//执行完一次iFileState循环后，控制器UsrData文件夹内有test2.txt文件，需要删除之后才能再次循环，否则重命名时因文件名已存在会报错	  
IF restart THEN
   DelFileName :='/usr/src/CODESYSControl/UsrData/test2.txt';
   xFileDelete:=TRUE;
   TON_2(IN:= xFileDelete, PT:= T#100MS, Q=> , ET=> );  //删除文件延时判断
      IF TON_2.Q THEN
		  IF FileDeleteErrorID = 0 THEN 
             xFileDelete :=FALSE;
             TON_2(IN:= xFileDelete, PT:= T#10MS, Q=> , ET=> );  //复位定时器
			 restart:=FALSE;
			 iFileState:=1;
			ELSE  xFileDelete:=FALSE;
                  iFileState:=10;
				  RETURN; 
		  END_IF  
	  END_IF 
END_IF         
END_CASE

ACTION ACT_SysFileRead:
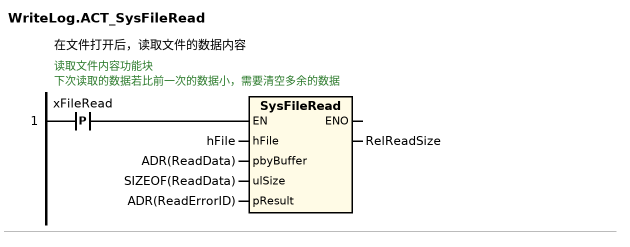
// NETWORK 1: 在文件打开后，读取文件的数据内容
// 读取文件内容功能块
// 下次读取的数据若比前一次的数据小，需要清空多余的数据
_rt1(CLK := xFileRead);
IF _rt1.Q THEN
    RelReadSize := SysFileRead(hFile := hFile, pbyBuffer := ADR(ReadData), ulSize := SIZEOF(ReadData), pResult := ADR(ReadErrorID));
END_IF
END_ACTION

ACTION ACT_SysFileDelete:
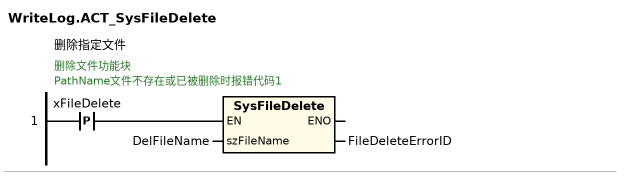
// NETWORK 1: 删除指定文件
// 删除文件功能块
// PathName文件不存在或已被删除时报错代码1
_rt2(CLK := xFileDelete);
IF _rt2.Q THEN FileDeleteErrorID := SysFileDelete(szFileName := DelFileName); END_IF
END_ACTION

ACTION ACT_SysFileClose:
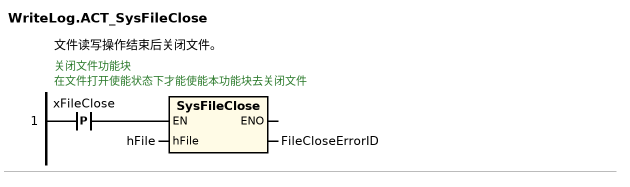
// NETWORK 1: 文件读写操作结束后关闭文件。
// 关闭文件功能块
// 在文件打开使能状态下才能使能本功能块去关闭文件
_rt3(CLK := xFileClose);
IF _rt3.Q THEN FileCloseErrorID := SysFileClose(hFile := hFile); END_IF
END_ACTION

ACTION ACT_SysFileRename:
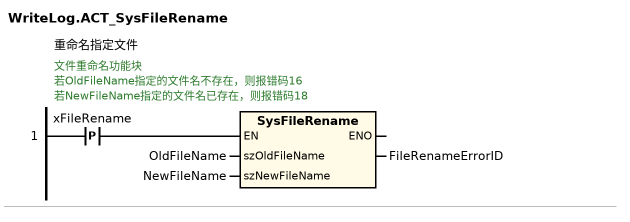
// NETWORK 1: 重命名指定文件
// 文件重命名功能块
// 若OldFileName指定的文件名不存在，则报错码16
// 若NewFileName指定的文件名已存在，则报错码18
_rt4(CLK := xFileRename);
IF _rt4.Q THEN
    FileRenameErrorID := SysFileRename(szOldFileName := OldFileName, szNewFileName := NewFileName);
END_IF
END_ACTION

ACTION ACT_SysFileGetPos:
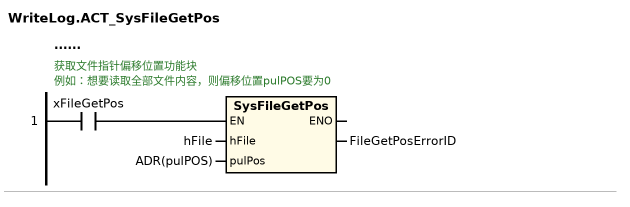
// NETWORK 1: ......
// 获取文件指针偏移位置功能块
// 例如：想要读取全部文件内容，则偏移位置pulPOS要为0
IF xFileGetPos THEN FileGetPosErrorID := SysFileGetPos(hFile := hFile, pulPos := ADR(pulPOS)); END_IF
END_ACTION

ACTION ACT_SysFileCopy:
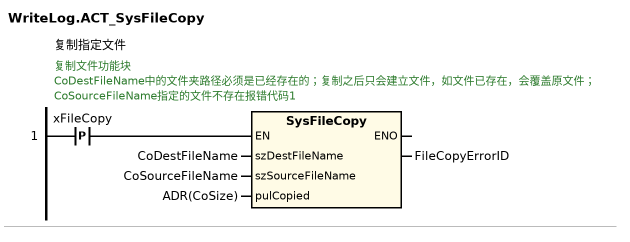
// NETWORK 1: 复制指定文件
// 复制文件功能块
// CoDestFileName中的文件夹路径必须是已经存在的；复制之后只会建立文件，如文件已存在，会覆盖原文件；
// CoSourceFileName指定的文件不存在报错代码1
_rt5(CLK := xFileCopy);
IF _rt5.Q THEN
    FileCopyErrorID := SysFileCopy(szDestFileName := CoDestFileName, szSourceFileName := CoSourceFileName, pulCopied := ADR(CoSize));
END_IF
END_ACTION

ACTION ACT_SysFileSetPos:
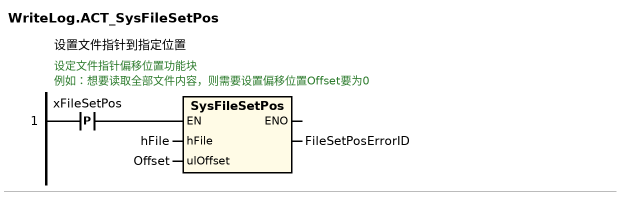
// NETWORK 1: 设置文件指针到指定位置
// 设定文件指针偏移位置功能块
// 例如：想要读取全部文件内容，则需要设置偏移位置Offset要为0
_rt6(CLK := xFileSetPos);
IF _rt6.Q THEN FileSetPosErrorID := SysFileSetPos(hFile := hFile, ulOffset := Offset); END_IF
END_ACTION

ACTION ACT_SysFileEOF:
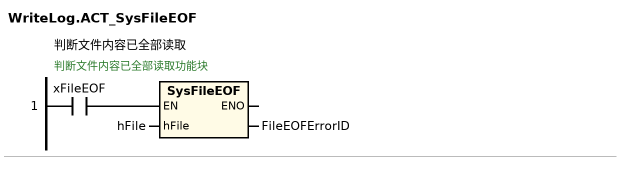
// NETWORK 1: 判断文件内容已全部读取
// 判断文件内容已全部读取功能块
IF xFileEOF THEN FileEOFErrorID := SysFileEOF(hFile := hFile); END_IF
END_ACTION

ACTION ACT_SysFileWrite:
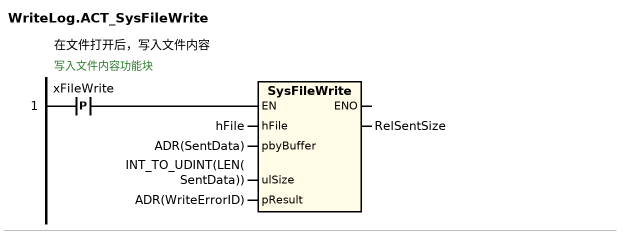
// NETWORK 1: 在文件打开后，写入文件内容
// 写入文件内容功能块
_rt7(CLK := xFileWrite);
IF _rt7.Q THEN
    RelSentSize := SysFileWrite(hFile := hFile, pbyBuffer := ADR(SentData), ulSize := INT_TO_UDINT(LEN(SentData)), pResult := ADR(WriteErrorID));
END_IF
END_ACTION

ACTION ACT_SysFileOpen:
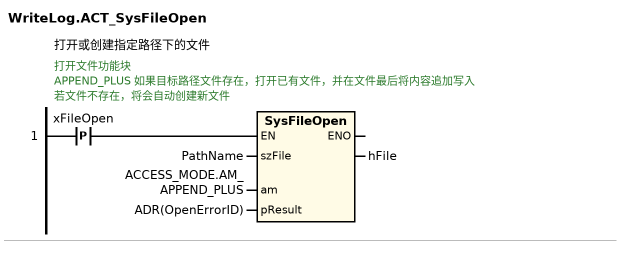
// NETWORK 1: 打开或创建指定路径下的文件
// 打开文件功能块
// APPEND_PLUS 如果目标路径文件存在，打开已有文件，并在文件最后将内容追加写入
//             若文件不存在，将会自动创建新文件
_rt8(CLK := xFileOpen);
IF _rt8.Q THEN
    hFile := SysFileOpen(szFile := PathName, am := ACCESS_MODE.AM_APPEND_PLUS, pResult := ADR(OpenErrorID));
END_IF
END_ACTION

END_PROGRAM

// Device/Application/BasicFBs/MeanValue
FUNCTION_BLOCK MeanValue
VAR_EXTERNAL

END_VAR

VAR_INPUT
	Input:UINT;
	PAR_Lenght:UINT;
	Reset:BOOL;
END_VAR
VAR_OUTPUT
	Output:UINT;
END_VAR
VAR
	Ka_Count:UINT:=1;
	Ka:UINT:=1;
	Ka_prev:UINT;
END_VAR

(*======================== READ_ME ==============================*)
(*功能块：“平均值滤波”                                         *)
(*=========================== END ===============================*)
	Ka:=UDINT_TO_UINT((UINT_TO_UDINT(Ka)*UINT_TO_UDINT(Ka_Count-1)+UINT_TO_UDINT(Input))/UINT_TO_UDINT(Ka_Count));
	Ka_Count:=Ka_count+1;
	IF(Reset OR Ka_count=PAR_Lenght+1) THEN
		Output:=Ka;
		Ka_Count:=1;
		Ka:=1;
	END_IF;

END_FUNCTION_BLOCK

// Device/Application/BasicFBs/Cut
FUNCTION_BLOCK Cut     (*把输入值进行预处理，调整斜率，消除两端的非线性影响*)
VAR_INPUT
	Input:UINT;
	PAR_InputlLowLimit:UINT;               (*此值的取值范围为0-255，一般在0—50之间*)
	PAR_InputHighLimit:UINT;               (*此值的取值范围为0-255，一般在200-255之间*)
END_VAR
VAR_OUTPUT
	Output:UINT;
	LowLimit:BOOL;
	HighLimit:BOOL;
END_VAR
VAR
END_VAR

(*功能描述：
把输入值进行预处理，调整斜率，消除两端非线性影响。
输入参数：
（1）Input，UINT型，要处理的信号。
（2）PAR_InputILowLimit，UINT型，用来控制输出的下限。当Input<=256*PAR_InputILowLimit时输出为0。
（3）PAR_InputHighLimit，UINT型，用来控制输出的上限。当Input>=256*PAR_InputHighLimit时输出就为256*PAR_InputHighLimit。
输出参数：
（1）Output，UINT型，处理完的信号。
（2）LowLimit，BOOL型，Input<=256*PAR_InputILowLimit时LowLimit为TRUE。
（3）HighLimit，BOOL型，Input>=256*PAR_InputHighLimit时HighLimit为TRUE。
*)

	LowLimit:=0;
	HighLimit:=0;
	PAR_InputlLowLimit:=PAR_InputlLowLimit*256;
	PAR_InputHighLimit:=PAR_InputHighLimit*256;
	IF(Input>=PAR_InputHighLimit) THEN
		Output:=0;
		HighLimit:=1;
	ELSIF(Input<=PAR_InputlLowLimit) THEN
		Output:=0;
		LowLimit:=1;
	ELSE
		Output:=DWORD_TO_UINT((Input-PAR_InputlLowLimit)*65536/(65536-PAR_InputlLowLimit-(65535-PAR_InputHighLimit)));
	END_IF

END_FUNCTION_BLOCK

// Device/Application/Motor
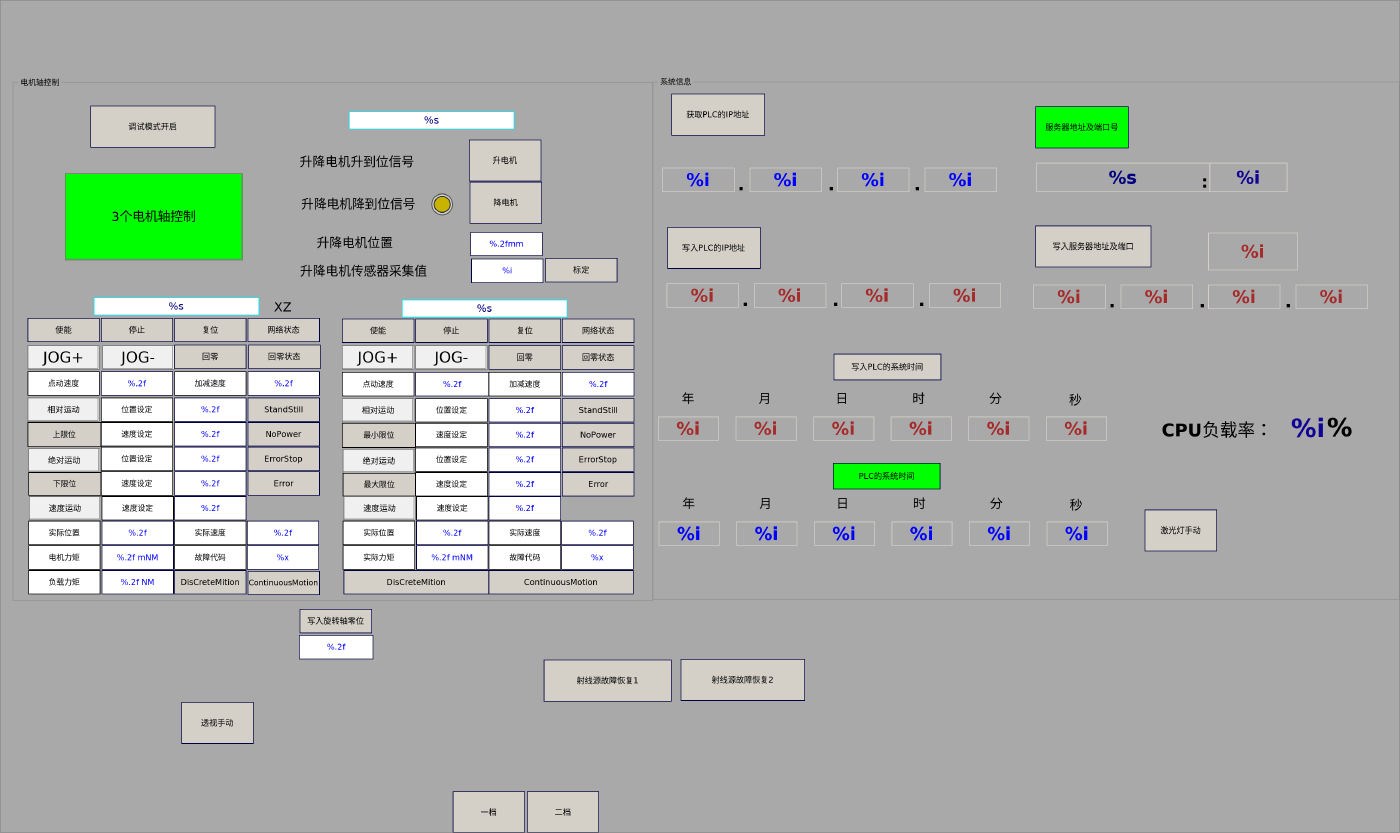
VISUALIZATION Motor  // 1985x1182
    Button (39,490 102x34), "JOG+", colour toggle: Axis_XZ.XZ_AxisCmd.bJogP
        tap Axis_XZ.XZ_AxisCmd.bJogP
    Rectangle (144,739 102x34), "%.2f", text variable: Axis_XZ.XZ_AxisState.rActPosition
    Button (145,490 102x34), "JOG-", colour toggle: Axis_XZ.XZ_AxisCmd.bJogN
        tap Axis_XZ.XZ_AxisCmd.bJogN
    RoundedRectangle (39,451 102x34), "使能", colour toggle: Axis_XZ.XZ_AxisState.bPowering
        toggle Axis_XZ.XZ_AxisCmd.bPower
    RoundedRectangle (351,451 102x34), "网络状态", colour toggle: Axis_XZ.XZ_AxisState.bNetState
    Button (40,636 102x34), "绝对运动", colour toggle: Axis_XZ.XZ_AxisCmd.bAbs
        tap Axis_XZ.XZ_AxisCmd.bAbs
    Rectangle (40,739 102x34), "实际位置"
    Rectangle (350,739 102x34), "%.2f", text variable: Axis_XZ.XZ_AxisState.rActVelocity
    Rectangle (247,739 102x34), "实际速度"
    RoundedRectangle (143,451 102x34), "停止", colour toggle: Axis_XZ.XZ_AxisState.bStopState
        tap Axis_XZ.XZ_AxisCmd.bStop
    RoundedRectangle (247,451 102x34), "复位", colour toggle: Axis_XZ.XZ_AxisCmd.bReset
        tap Axis_XZ.XZ_AxisCmd.bReset
    Rectangle (133,422 234x25), "%s", text variable: InitMotor.sNameXZ, text list: ''
    Rectangle (247,774 102x34), "故障代码"
    Rectangle (350,774 102x34), "%x", text variable: Axis_XZ.XZ_AxisState.ErrorID, colour toggle: (Axis_XZ.XZ_AxisState.ErrorID)<>0
    Rectangle (40,670 103x33), "下限位", colour toggle: Entity_IO.bRotateMotorMin
    Rectangle (39,599 104x35), "上限位", colour toggle: Entity_IO.bRotateMotorMax
    RoundedRectangle (247,489 102x34), "回零", colour toggle: Axis_XZ.XZ_AxisCmd.bHome
        tap Axis_XZ.XZ_AxisCmd.bHome
    Button (39,564 102x34), "相对运动", colour toggle: Axis_XZ.XZ_AxisCmd.bRel
        tap Axis_XZ.XZ_AxisCmd.bRel
    Rectangle (143,527 102x34), "%.2f", text variable: Axis_XZ.XZ_AxisCmd.AxisPara.rJogVelocity
        OnMouseClick: write Axis_XZ.XZ_AxisCmd.AxisPara.rJogVelocity via Default
    Rectangle (39,527 102x34), "点动速度"
    Rectangle (247,527 102x34), "加减速度"
    Rectangle (351,527 102x34), "%.2f", text variable: Axis_XZ.XZ_AxisCmd.AxisPara.rAccDec
        OnMouseClick: write Axis_XZ.XZ_AxisCmd.AxisPara.rAccDec via Default
    Rectangle (143,564 102x34), "位置设定"
    Rectangle (247,564 102x34), "%.2f", text variable: Axis_XZ.XZ_AxisCmd.AxisPara.rRelPosition
        OnMouseClick: write Axis_XZ.XZ_AxisCmd.AxisPara.rRelPosition via Default
    Rectangle (143,599 102x34), "速度设定"
    Rectangle (247,599 102x34), "%.2f", text variable: Axis_XZ.XZ_AxisCmd.AxisPara.rRelVelocity
        OnMouseClick: write Axis_XZ.XZ_AxisCmd.AxisPara.rRelVelocity via Default
    Rectangle (143,634 102x34), "位置设定"
    Rectangle (693,635 102x34), "%.2f", text variable: Axis_QJ.QJ_AxisCmd.AxisPara.rAbsPosition
        OnMouseClick: write Axis_QJ.QJ_AxisCmd.AxisPara.rAbsPosition via Default
    Rectangle (143,669 102x34), "速度设定"
    Rectangle (247,669 102x34), "%.2f", text variable: Axis_XZ.XZ_AxisCmd.AxisPara.rAbsVelocity
        OnMouseClick: write Axis_XZ.XZ_AxisCmd.AxisPara.rAbsVelocity via Default
    RoundedRectangle (351,564 102x34), "StandStill", colour toggle: Axis_XZ.XZ_AxisState.bStandStill
    RoundedRectangle (351,599 102x34), "NoPower", colour toggle: Axis_XZ.XZ_AxisState.bPowerOff
    RoundedRectangle (351,634 102x34), "ErrorStop", colour toggle: Axis_XZ.XZ_AxisState.bErrStop
    RoundedRectangle (351,669 102x34), "Error", colour toggle: Axis_XZ.XZ_AxisState.bAxisErr
    Rectangle (144,774 102x34), "%.2f mNM", text variable: Axis_XZ.XZ_AxisState.rActTorque
    Rectangle (40,774 102x34), "电机力矩"
    Rectangle (570,425 234x25), "%s", text variable: InitMotor.sNameQJ, text list: ''
    Button (485,490 102x34), "JOG+", colour toggle: Axis_QJ.QJ_AxisCmd.bJogP
        tap Axis_QJ.QJ_AxisCmd.bJogP
    Rectangle (590,739 102x34), "%.2f", text variable: Axis_QJ.QJ_AxisState.rActPosition
    Button (589,490 102x34), "JOG-", colour toggle: Axis_QJ.QJ_AxisCmd.bJogN
        tap Axis_QJ.QJ_AxisCmd.bJogN
    RoundedRectangle (485,452 102x34), "使能", colour toggle: Axis_QJ.QJ_AxisState.bPowering
        toggle Axis_QJ.QJ_AxisCmd.bPower
    RoundedRectangle (797,452 102x34), "网络状态", colour toggle: Axis_QJ.QJ_AxisState.bNetState
    Button (486,637 102x34), "绝对运动", colour toggle: Axis_QJ.QJ_AxisCmd.bAbs
        tap Axis_QJ.QJ_AxisCmd.bAbs
    Rectangle (486,739 102x34), "实际位置"
    Rectangle (796,739 102x34), "%.2f", text variable: Axis_QJ.QJ_AxisState.rActVelocity
    Rectangle (693,739 102x34), "实际速度"
    RoundedRectangle (589,452 102x34), "停止", colour toggle: Axis_QJ.QJ_AxisCmd.bStop
        tap Axis_QJ.QJ_AxisCmd.bStop
    RoundedRectangle (693,452 102x34), "复位", colour toggle: Axis_QJ.QJ_AxisCmd.bReset
        tap Axis_QJ.QJ_AxisCmd.bReset
    Rectangle (693,774 102x34), "故障代码"
    Rectangle (796,774 102x34), "%x", text variable: Axis_QJ.QJ_AxisState.ErrorID, colour toggle: (Axis_QJ.QJ_AxisState.ErrorID)<>0
    Rectangle (486,671 103x33), "最大限位", colour toggle: Entity_IO.bForeMotorMax
    Rectangle (485,600 104x35), "最小限位", colour toggle: Entity_IO.bForeMotorMin
    RoundedRectangle (693,490 102x34), "回零", colour toggle: Axis_QJ.QJ_AxisCmd.bHome
        tap Axis_QJ.QJ_AxisCmd.bHome
    Button (485,565 102x34), "相对运动", colour toggle: Axis_QJ.QJ_AxisCmd.bRel
        tap Axis_QJ.QJ_AxisCmd.bRel
    Rectangle (589,528 104x34), "%.2f", text variable: Axis_QJ.QJ_AxisCmd.AxisPara.rJogVelocity
        OnMouseClick: write Axis_QJ.QJ_AxisCmd.AxisPara.rJogVelocity via Default
    Rectangle (485,528 102x34), "点动速度"
    Rectangle (693,528 102x34), "加减速度"
    Rectangle (797,528 102x34), "%.2f", text variable: Axis_QJ.QJ_AxisCmd.AxisPara.rAccDec
        OnMouseClick: write Axis_QJ.QJ_AxisCmd.AxisPara.rAccDec via Default
    Rectangle (589,565 102x34), "位置设定"
    Rectangle (693,565 102x34), "%.2f", text variable: Axis_QJ.QJ_AxisCmd.AxisPara.rRelPosition
        OnMouseClick: write Axis_QJ.QJ_AxisCmd.AxisPara.rRelPosition via Default, min -1000, max 1000
    Rectangle (589,600 102x34), "速度设定"
    Rectangle (693,600 102x34), "%.2f", text variable: Axis_QJ.QJ_AxisCmd.AxisPara.rRelVelocity
        OnMouseClick: write Axis_QJ.QJ_AxisCmd.AxisPara.rRelVelocity via Default
    Rectangle (589,635 102x34), "位置设定"
    Rectangle (247,634 102x34), "%.2f", text variable: Axis_XZ.XZ_AxisCmd.AxisPara.rAbsPosition
        OnMouseClick: write Axis_XZ.XZ_AxisCmd.AxisPara.rAbsPosition via Default
    Rectangle (589,670 102x34), "速度设定"
    Rectangle (693,670 102x34), "%.2f", text variable: Axis_QJ.QJ_AxisCmd.AxisPara.rAbsVelocity
        OnMouseClick: write Axis_QJ.QJ_AxisCmd.AxisPara.rAbsVelocity via Default
    RoundedRectangle (797,565 102x34), "StandStill", colour toggle: Axis_QJ.QJ_AxisState.bStandStill
    RoundedRectangle (797,600 102x34), "NoPower", colour toggle: Axis_QJ.QJ_AxisState.bPowerOff
    RoundedRectangle (797,635 102x34), "ErrorStop", colour toggle: Axis_QJ.QJ_AxisState.bErrStop
    RoundedRectangle (797,670 102x34), "Error", colour toggle: Axis_QJ.QJ_AxisState.bAxisErr
    Rectangle (590,774 102x34), "%.2f mNM", text variable: Axis_QJ.QJ_AxisState.rActTorque
    Rectangle (486,774 102x34), "实际力矩"
    RoundedRectangle (487,809 206x34), "DisCreteMition", colour toggle: Axis_QJ.QJ_AxisState.bDisCreteMition
    RoundedRectangle (693,809 205x34), "ContinuousMotion", colour toggle: Axis_QJ.QJ_AxisState.bContinuousMotion
    RoundedRectangle (247,809 102x34), "DisCreteMition", colour toggle: Axis_XZ.XZ_AxisState.bDisCreteMition
    RoundedRectangle (351,810 102x34), "ContinuousMotion", colour toggle: Axis_XZ.XZ_AxisState.bContinuousMotion
    RoundedRectangle (128,150 177x59), "调试模式开启", colour toggle: WorkMode.bDebugMode
        toggle WorkMode.bDebugMode
    Rectangle (495,158 234x25), "%s", text variable: InitMotor.sNameSJ, text list: ''
    RoundedRectangle (665,198 102x59), "升电机", colour toggle: Entity_IO.bUpMotorPos
        tap Entity_IO.bUpMotorPos
    RoundedRectangle (666,258 102x59), "降电机", colour toggle: Entity_IO.bUpMotorNeg
        tap Entity_IO.bUpMotorNeg
    Label (410,212 192x36), "升降电机升到位信号"
    Label (412,272 192x36), "升降电机降到位信号"
    Lamp1 (608,272 38x36), variable: Entity_IO.bUpMotorMin, style: Lamp-Lamp1-Yellow
    Button (92,246 252x123), "3个电机轴控制"
        OnMouseClick:  Assign=Catalogue, Type=Assignment
    RoundedRectangle (773,366 102x34), "标定", colour toggle: Entity_IO.bCalibrate
        tap Entity_IO.bCalibrate
    Rectangle (667,329 102x34), "%.2fmm", text variable: Entity_IO.rRealPos
        OnMouseClick: write  via Default, min -100, max 1000
    Label (407,327 192x36), "升降电机位置"
    Rectangle (668,367 102x34), "%i", text variable: Entity_IO.AIX0
        OnMouseClick: write  via Default, min -100, max 1000
    Label (386,367 259x36), "升降电机传感器采集值"
    RoundedRectangle (352,489 102x34), "回零状态", colour toggle: Axis_XZ.XZ_AxisState.bHoming
    RoundedRectangle (797,490 102x34), "回零状态", colour toggle: Axis_QJ.QJ_AxisState.bHoming
    Rectangle (939,238 102x34), "%i", text variable: PLC_PRG.LS_GetIPAddress_1.byIpSegmengt1
    Label (1033,248 36x26), "."
    Label (1161,248 36x26), "."
    Label (1283,248 36x26), "."
    Rectangle (1063,238 102x34), "%i", text variable: PLC_PRG.LS_GetIPAddress_1.byIpSegmengt2
    Rectangle (1187,238 102x34), "%i", text variable: PLC_PRG.LS_GetIPAddress_1.byIpSegmengt3
    Rectangle (1311,238 102x34), "%i", text variable: PLC_PRG.LS_GetIPAddress_1.byIpSegmengt4
    RoundedRectangle (946,322 132x59), "写入PLC的IP地址", colour toggle: PLC_PRG.bSetPLC_IP
        tap PLC_PRG.bSetPLC_IP
    Rectangle (945,402 102x34), "%i", text variable: PLC_PRG.LS_SetIPAddress_1.byIpSegmengt1
        OnMouseClick: write PLC_PRG.LS_SetIPAddress_1.byIpSegmengt1 via Default, min 0, max 1000
    Label (1039,412 36x26), "."
    Label (1167,412 36x26), "."
    Label (1289,412 36x26), "."
    Rectangle (1069,402 102x34), "%i", text variable: PLC_PRG.LS_SetIPAddress_1.byIpSegmengt2
        OnMouseClick: write PLC_PRG.LS_SetIPAddress_1.byIpSegmengt2 via Default, min 0, max 1000
    Rectangle (1193,402 102x34), "%i", text variable: PLC_PRG.LS_SetIPAddress_1.byIpSegmengt3
        OnMouseClick: write PLC_PRG.LS_SetIPAddress_1.byIpSegmengt3 via Default, min 0, max 1000
    Rectangle (1317,402 102x34), "%i", text variable: PLC_PRG.LS_SetIPAddress_1.byIpSegmengt4
        OnMouseClick: write PLC_PRG.LS_SetIPAddress_1.byIpSegmengt4 via Default, min 0, max 1000
    Rectangle (1817,583 76x49), "%i", text variable: PLC_PRG.rPLC_Load
    Label (1630,592 192x36), "CPU负载率："
    Label (1865,584 69x45), "%"
    Rectangle (933,591 86x34), "%i", text variable: PLC_PRG.LS_SetDintDT_1.uiYear
        OnMouseClick: write PLC_PRG.LS_SetDintDT_1.uiYear via Default, min 0, max 10000
    Rectangle (1043,591 86x34), "%i", text variable: PLC_PRG.LS_SetDintDT_1.uiMonth
        OnMouseClick: write PLC_PRG.LS_SetDintDT_1.uiMonth via Default, min 0, max 1000
    Rectangle (1153,591 86x34), "%i", text variable: PLC_PRG.LS_SetDintDT_1.uiDay
        OnMouseClick: write PLC_PRG.LS_SetDintDT_1.uiDay via Default, min 0, max 1000
    Rectangle (1263,591 86x34), "%i", text variable: PLC_PRG.LS_SetDintDT_1.uiHour
        OnMouseClick: write PLC_PRG.LS_SetDintDT_1.uiHour via Default, min 0, max 1000
    Rectangle (1373,591 86x34), "%i", text variable: PLC_PRG.LS_SetDintDT_1.uiMinute
        OnMouseClick: write PLC_PRG.LS_SetDintDT_1.uiMinute via Default, min 0, max 1000
    Rectangle (1483,591 86x34), "%i", text variable: PLC_PRG.LS_SetDintDT_1.uiSecond
        OnMouseClick: write PLC_PRG.LS_SetDintDT_1.uiSecond via Default, min 0, max 1000
    Label (942,548 67x36), "年"
    Label (1051,548 67x36), "月"
    Label (1160,548 67x36), "日"
    Label (1269,548 67x36), "时"
    Label (1378,548 67x36), "分"
    Label (1491,550 67x36), "秒"
    RoundedRectangle (1182,502 152x37), "写入PLC的系统时间", colour toggle: PLC_PRG.bSetSysTime
        tap PLC_PRG.bSetSysTime
    Rectangle (934,740 86x34), "%i", text variable: PLC_PRG.LS_ReadDintDT_1.uiYear
    Rectangle (1044,740 86x34), "%i", text variable: PLC_PRG.LS_ReadDintDT_1.uiMonth
    Rectangle (1154,740 86x34), "%i", text variable: PLC_PRG.LS_ReadDintDT_1.uiDay
    Rectangle (1264,740 86x34), "%i", text variable: PLC_PRG.LS_ReadDintDT_1.uiHour
    Rectangle (1374,740 86x34), "%i", text variable: PLC_PRG.LS_ReadDintDT_1.uiMinute
    Rectangle (1484,740 86x34), "%i", text variable: PLC_PRG.LS_ReadDintDT_1.uiSecond
    Label (943,697 67x36), "年"
    Label (1052,697 67x36), "月"
    Label (1161,697 67x36), "日"
    Label (1270,697 67x36), "时"
    Label (1379,697 67x36), "分"
    Label (1492,699 67x36), "秒"
    RoundedRectangle (1181,657 152x37), "PLC的系统时间"
    GroupBox (18,109 908x743), "电机轴控制"
        Label (287,309 192x36), "XZ"
    GroupBox (925,108 1060x743), "系统信息"
        RoundedRectangle (698,615 102x59), "激光灯手动", colour toggle: PLC_PRG.bDebug_Laser
            toggle PLC_PRG.bDebug_Laser
    Rectangle (1469,231 246x41), "%s", text variable: WorkStation_TCP.IP.sAddr, text list: ''
    Rectangle (1715,231 110x41), "%i", text variable: WorkStation_TCP.TCP_Client_1.uiPort
    Label (1685,239 46x37), ":"
    RoundedRectangle (1468,151 132x59), "服务器地址及端口号"
    RoundedRectangle (1468,320 164x59), "写入服务器地址及端口", colour toggle: WorkStation_TCP.bSetServerIP
        tap WorkStation_TCP.bSetServerIP
    Rectangle (1465,404 102x34), "%i", text variable: WorkStation_TCP.iServerIP1
        OnMouseClick: write WorkStation_TCP.iServerIP1 via Default, min 0, max 1000
    Label (1559,414 36x26), "."
    Label (1687,414 36x26), "."
    Label (1809,414 36x26), "."
    Rectangle (1589,404 102x34), "%i", text variable: WorkStation_TCP.iServerIP2
        OnMouseClick: write WorkStation_TCP.iServerIP2 via Default, min 0, max 1000
    Rectangle (1713,404 102x34), "%i", text variable: WorkStation_TCP.iServerIP3
        OnMouseClick: write WorkStation_TCP.iServerIP3 via Default, min 0, max 1000
    Rectangle (1837,404 102x34), "%i", text variable: WorkStation_TCP.iServerIP4
        OnMouseClick: write WorkStation_TCP.iServerIP4 via Default, min 0, max 1000
    Rectangle (1713,330 127x53), "%i", text variable: WorkStation_TCP.ServeruiPort
        OnMouseClick: write WorkStation_TCP.ServeruiPort via Default, min 0, max 65535
    Button (41,704 102x34), "速度运动", colour toggle: Axis_XZ.XZ_AxisCmd.bVel
        tap Axis_XZ.XZ_AxisCmd.bVel
    Rectangle (144,704 102x34), "速度设定"
    Rectangle (247,704 102x34), "%.2f", text variable: Axis_XZ.XZ_AxisCmd.AxisPara.rVelVelocity
        OnMouseClick: write Axis_XZ.XZ_AxisCmd.AxisPara.rVelVelocity via Default
    Button (487,704 102x34), "速度运动", colour toggle: Axis_QJ.QJ_AxisCmd.bVel
        tap Axis_QJ.QJ_AxisCmd.bVel
    Rectangle (590,704 102x34), "速度设定"
    Rectangle (693,704 102x34), "%.2f", text variable: Axis_QJ.QJ_AxisCmd.AxisPara.rVelVelocity
        OnMouseClick: write Axis_QJ.QJ_AxisCmd.AxisPara.rVelVelocity via Default
    Rectangle (144,809 102x34), "%.2f NM", text variable: Axis_XZ.rLoadTorque
    Rectangle (40,809 102x34), "负载力矩"
    RoundedRectangle (952,133 132x59), "获取PLC的IP地址", colour toggle: PLC_PRG.bGetPLC_IP
        tap PLC_PRG.bGetPLC_IP
    RoundedRectangle (425,864 102x34), "写入旋转轴零位", colour toggle: Entity_IO.bCalibrate
        tap Entity_IO.bCalibrate
    Rectangle (424,901 105x34), "%.2f", text variable: GVL_Retain.rXZ_Zero
        OnMouseClick: write GVL_Retain.rXZ_Zero via Default
    RoundedRectangle (771,936 181x59), "射线源故障恢复1", colour toggle: DT_Xray.bResetXray1
        tap DT_Xray.bResetXray1
    RoundedRectangle (965,935 176x59), "射线源故障恢复2", colour toggle: DT_Xray.bResetXray2
        tap DT_Xray.bResetXray2
    RoundedRectangle (257,996 102x59), "透视手动", colour toggle: Entity_IO.bXaryFlu
        toggle PLC_PRG.bTestFLU
    RoundedRectangle (642,1123 102x59), "一档", colour toggle: Entity_IO.bXaryOne
        toggle PLC_PRG.bbb
    RoundedRectangle (747,1123 102x59), "二档", colour toggle: Entity_IO.bXaryTwo
        toggle PLC_PRG.ccc
END_VISUALIZATION

// Device/Application/Entity_IO
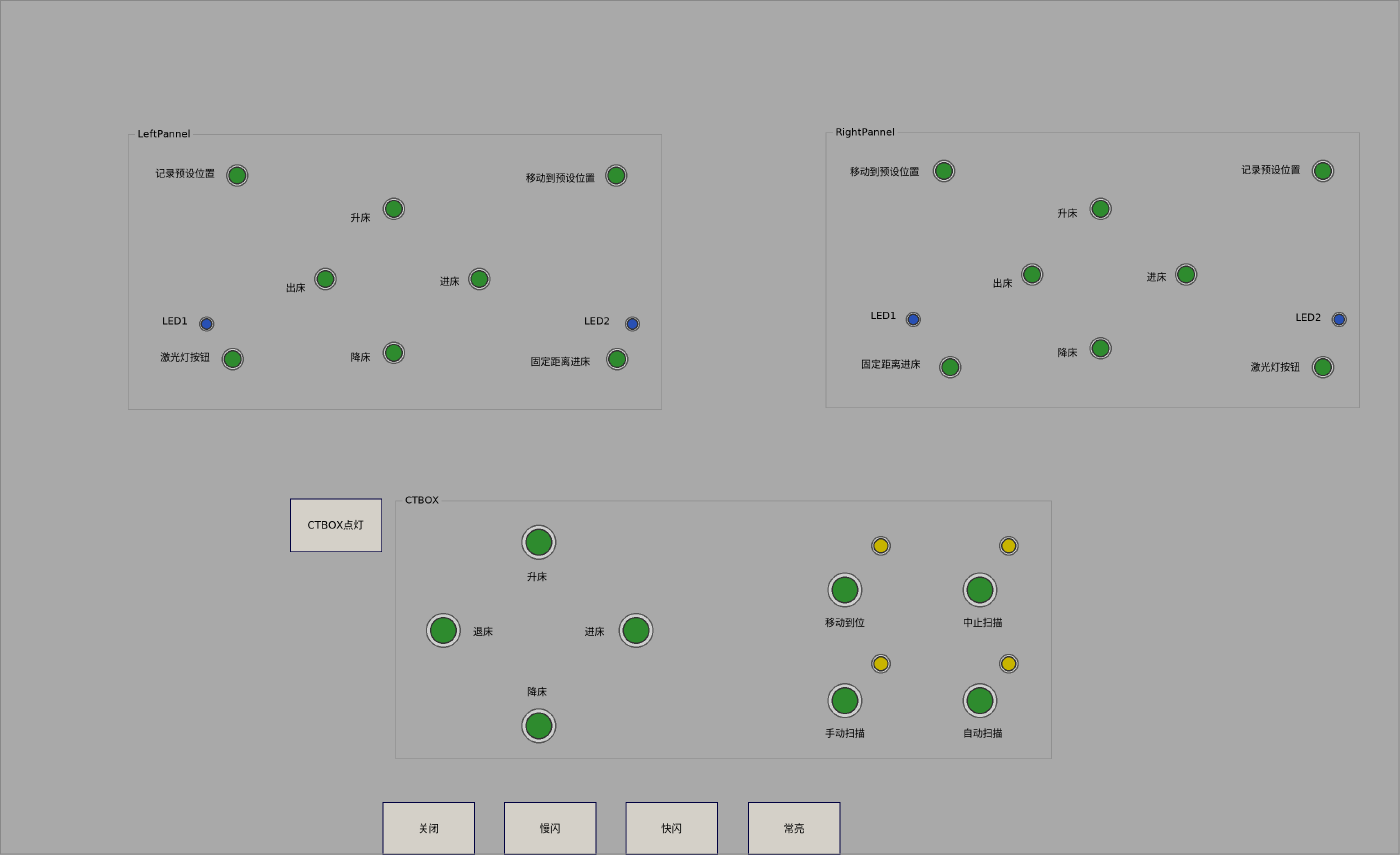
VISUALIZATION Entity_IO  // 1555x950
    Label (104,379 203x36), "激光灯按钮"
    Label (104,175 203x36), "记录预设位置"
    Lamp1 (423,217 29x30), variable: Entity_IO.LeftPannel_BedUp, style: Lamp-Lamp1-Green
    Lamp1 (423,377 29x30), variable: Entity_IO.LeftPannel_BedDown, style: Lamp-Lamp1-Green
    Label (299,379 203x36), "降床"
    Label (521,384 203x36), "固定距离进床"
    Label (227,302 203x36), "出床"
    Label (299,224 203x36), "升床"
    Label (398,295 203x36), "进床"
    Label (521,180 203x36), "移动到预设位置"
    Lamp1 (347,295 29x30), variable: Entity_IO.LeftPannel_BedBack, style: Lamp-Lamp1-Green
    Lamp1 (518,295 29x30), variable: Entity_IO.LeftPannel_BedFore, style: Lamp-Lamp1-Green
    Lamp1 (244,384 29x30), variable: Entity_IO.LeftPannel_LaserButton, style: Lamp-Lamp1-Green
    Lamp1 (249,180 29x30), variable: Entity_IO.LeftPannel_RecordPos, style: Lamp-Lamp1-Green
    Lamp1 (671,384 29x30), variable: Entity_IO.LeftPannel_DistanceMove, style: Lamp-Lamp1-Green
    Lamp1 (670,180 29x30), variable: Entity_IO.LeftPannel_MoveRecordPos, style: Lamp-Lamp1-Green
    Lamp1 (693,349 19x22), variable: Entity_IO.bLeftPannel_LED2, style: Lamp-Lamp1-Blue
    Lamp1 (220,349 19x22), variable: Entity_IO.bLeftPannel_LED1, style: Lamp-Lamp1-Blue
    Label (562,339 203x36), "LED2"
    Label (93,339 203x36), "LED1"
    Lamp1 (1208,372 29x30), variable: Entity_IO.RightPannel_BedDown, style: Lamp-Lamp1-Green
    Label (1084,374 203x36), "降床"
    Label (888,387 203x36), "固定距离进床"
    Label (1012,297 203x36), "出床"
    Label (1315,390 203x36), "激光灯按钮"
    Label (1310,171 203x36), "记录预设位置"
    Label (1084,219 203x36), "升床"
    Label (1183,290 203x36), "进床"
    Label (881,173 203x36), "移动到预设位置"
    Lamp1 (1132,290 29x30), variable: Entity_IO.RightPannel_BedBack, style: Lamp-Lamp1-Green
    Lamp1 (1303,290 29x30), variable: Entity_IO.RightPannel_BedFore, style: Lamp-Lamp1-Green
    Lamp1 (1455,393 29x30), variable: Entity_IO.RightPannel_LaserButton, style: Lamp-Lamp1-Green
    Lamp1 (1034,175 29x30), variable: Entity_IO.RightPannel_MoveRecordPos, style: Lamp-Lamp1-Green
    Lamp1 (1041,393 29x30), variable: Entity_IO.RightPannel_DistanceMove, style: Lamp-Lamp1-Green
    Lamp1 (1455,175 29x30), variable: Entity_IO.RightPannel_RecordPos, style: Lamp-Lamp1-Green
    Lamp1 (1478,344 19x22), variable: Entity_IO.bRightPannel_LED2, style: Lamp-Lamp1-Blue
    Lamp1 (1005,344 19x22), variable: Entity_IO.bRightPannel_LED1, style: Lamp-Lamp1-Blue
    Label (1352,335 203x36), "LED2"
    Label (880,333 203x36), "LED1"
    Lamp1 (1208,217 29x30), variable: Entity_IO.RightPannel_BedUp, style: Lamp-Lamp1-Green
    Lamp1 (576,580 45x45), variable: CTBOX_RS232.CTBOX_KEY[5], style: Lamp-Lamp1-Green
    Lamp1 (576,784 45x45), variable: CTBOX_RS232.CTBOX_KEY[7], style: Lamp-Lamp1-Green
    Lamp1 (684,678 45x45), variable: CTBOX_RS232.CTBOX_KEY[4], style: Lamp-Lamp1-Green
    Lamp1 (470,678 45x45), variable: CTBOX_RS232.CTBOX_KEY[6], style: Lamp-Lamp1-Green
    Lamp1 (916,633 45x45), variable: CTBOX_RS232.CTBOX_KEY[3], style: Lamp-Lamp1-Green
    Lamp1 (1066,633 45x45), variable: CTBOX_RS232.CTBOX_KEY[2], style: Lamp-Lamp1-Green
    Lamp1 (916,756 45x45), variable: CTBOX_RS232.CTBOX_KEY[0], style: Lamp-Lamp1-Green
    Lamp1 (1066,756 45x45), variable: CTBOX_RS232.CTBOX_KEY[1], style: Lamp-Lamp1-Green
    Lamp1 (966,725 25x25), variable: CTBOX_RS232.Lamp7State<>0, style: Lamp-Lamp1-Yellow
    Lamp1 (1108,725 25x25), variable: CTBOX_RS232.Lamp8State<>0, style: Lamp-Lamp1-Yellow
    Lamp1 (966,594 25x25), variable: CTBOX_RS232.Lamp5State<>0, style: Lamp-Lamp1-Yellow
    Lamp1 (1108,594 25x25), variable: CTBOX_RS232.Lamp6State<>0, style: Lamp-Lamp1-Yellow
    GroupBox (142,141 593x314), "LeftPannel"
    GroupBox (917,139 593x314), "RightPannel"
    GroupBox (439,548 729x295), "CTBOX"
    Label (515,623 163x36), "升床"
    Label (515,751 163x36), "降床"
    Label (455,684 163x36), "退床"
    Label (579,684 163x36), "进床"
    Label (857,674 163x36), "移动到位"
    Label (1010,674 163x36), "中止扫描"
    Label (857,797 163x36), "手动扫描"
    Label (1010,797 163x36), "自动扫描"
    RoundedRectangle (322,554 102x59), "CTBOX点灯", colour toggle: CTBOX_RS232.bDebug_RS232
        toggle CTBOX_RS232.bDebug_RS232
    RoundedRectangle (425,891 102x59), "关闭", colour toggle: CTBOX_RS232.A1
        toggle CTBOX_RS232.A1
    RoundedRectangle (560,891 102x59), "慢闪", colour toggle: CTBOX_RS232.A2
        toggle CTBOX_RS232.A2
    RoundedRectangle (695,891 102x59), "快闪", colour toggle: CTBOX_RS232.A3
        toggle CTBOX_RS232.A3
    RoundedRectangle (831,891 102x59), "常亮", colour toggle: CTBOX_RS232.A4
        toggle CTBOX_RS232.A4
END_VISUALIZATION
